% RSLogix 500 project practice3.RSS, saved by version 8.30.00.16 %
PROJECT "UNTITLED"    % processor: Bul.1763 MicroLogix 1100 Series B %

PROGRAM FILES
  LAD 2   6 rungs

DATA FILES
  O0 OUTPUT  4 elements
  I1 INPUT  6 elements
  S2 STATUS  66 elements
  B3 BINARY  1 elements
  T4 TIMER  1 elements
  C5 COUNTER  1 elements
  R6 CONTROL  1 elements
  N7 INTEGER  1 elements
  F8 FLOAT  1 elements

LADDER 2
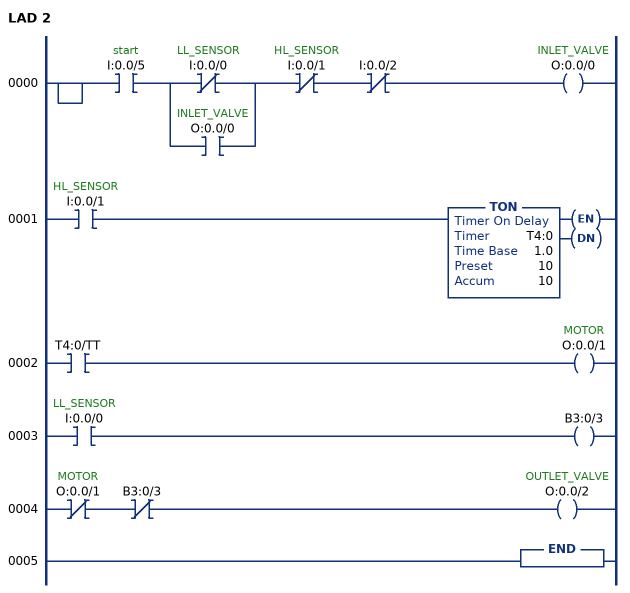
% Rung: 0 %
SOR BST NXB BND XIC I:0.0/5 BST XIO I:0.0/0 NXB XIC O:0.0/0 BND XIO I:0.0/1 XIO I:0.0/2 OTE O:0.0/0 EOR
%   I:0.0/5  "start" %
%   I:0.0/0  "LL_SENSOR" %
%   O:0.0/0  "INLET_VALVE" %
%   I:0.0/1  "HL_SENSOR" %
% Rung: 1 %
SOR XIC I:0.0/1 TON T4:0 1.0 10 10 EOR
%   I:0.0/1  "HL_SENSOR" %
% Rung: 2 %
SOR XIC T4:0/TT OTE O:0.0/1 EOR
%   O:0.0/1  "MOTOR" %
% Rung: 3 %
SOR XIC I:0.0/0 OTE B3:0/3 EOR
%   I:0.0/0  "LL_SENSOR" %
% Rung: 4 %
SOR XIO O:0.0/1 XIO B3:0/3 OTE O:0.0/2 EOR
%   O:0.0/1  "MOTOR" %
%   O:0.0/2  "OUTLET_VALVE" %
% Rung: 5 %
SOR END EOR

OTHER DOCUMENTED ADDRESSES
  I:0.0/4  "lOW lAVEL"

DATA TABLE (non-zero values as saved)
DATA T4
% .PRE .ACC %
% T4:0 % 10 10
